Staubli VAL3: MainProg1.pjx

--- MainProg1.pjx ---
Parameters version=s7.3.1 stackSize=5000 millimeterUnit=true
Program file=loadNextOne.pgx
Program file=start.pgx
Program file=stop.pgx
Data file=MainProg1.dtx
Library alias=prog path=./Prog1/Prog1.pjx
Library alias=prog_swap path=./Prog1/Prog1.pjx
Library alias=tooldata path=saveChangeTool

--- MainProg1.dtx ---
public dio dioIN = {link=fIn0}
public dio dioOUT = {link=fOut0}
public dio dioRotationON = {link=BasicIO-1\%Q0}
public dio dioRotationOFF = {link=BasicIO-1\%Q1}
public dio dioBuse = {link=BasicIO-1\%Q2}
public frame fPartCad = {x=0.000, y=0.000, z=0.000, rx=-0.000, ry=0.000, rz=-0.000, fatherId=world[0]}
public frame fCadToReal = {x=0, y=0, z=0, rx=0, ry=0, rz=0, fatherId=fPartCad[0]}
public mdesc mNomSpeed = {accel=100, vel=100, decel=100, tmax=99999, rmax=99999, blend=off, leave=50, reach=50}
public num nTraj
num nTimeStop
num nTimeStart
num nMode
num nEtat
public tool tCad = {x=0.000, y=0.000, z=0.000, rx=0.000, ry=0.000, rz=0.000, fatherId=flange[0], ioLink=valve1}

--- start.pgx ---
public program start()
begin
  if prog:libLoad("./Prog1")!=0
    logMsg("Error Loading RoboDK library")
    popUpMsg("Error Loading RoboDK library")
  endIf
  wait(taskStatus("loading")==-1)
  prog:fPartReal.trsf=fPartCad.trsf*fCadToReal.trsf
  prog:tCad.trsf=prog:tCad.trsf*{0,0,tooldata:nLength,0,0,0}
  call prog:start()


end

--- loadNextOne.pgx ---
program loadNextOne(string x_sName)
begin
  prog_swap:libLoad(x_sName)
end
